{attribute 'qualified_only'}
VAR_GLOBAL
	bDigital_Inputs AT %I* : ARRAY[1..8] OF BOOL;
	bDigital_Outputs AT %Q* : ARRAY[1..8] OF BOOL;
END_VAR

(* stored: Version 1.1.0.1, ProductVersion 3.1.4024.12
   GVL GVL: Id {2cfc2c01-fbfe-4516-966b-defb3309a9f1} *)
